// TwinCAT 3 PLC project Untitled1
// ProgramVersion: 3.1.4024.0
// libraries:
//   Tc2_MC2, * (Beckhoff Automation GmbH)
//   Tc2_Standard, * (Beckhoff Automation GmbH)
//   Tc2_System, * (Beckhoff Automation GmbH)
//   Tc2_Utilities, * (Beckhoff Automation GmbH)
//   Tc3_Module, * (Beckhoff Automation GmbH)
//   VisuDialogs, * (System)
// project tree:
//   / GlobalTextList.TcGTLO, PlcTask.TcTTO, Visualization Manager.TcVMO (not stored), VISU_TASK.TcTTO
//   POUs/ACTION/ E_ACTION_STATE.TcDUT, FB_ACTION.TcPOU, vACTION.TcVIS
//   POUs/AXES/ AXES_CYCLE.TcPOU, FB_Axis.TcPOU, GVL_AXES.TcGVL, vAXIS.TcVIS
//   POUs/EVENT_LOGGER/ E_EventType.TcDUT (not stored), FB_EventLogger.TcPOU (not stored), GVL_EVENT_LOGGER.TcGVL (not stored), ST_Event.TcDUT (not stored), UpdateEventTimestampWithSystemTime.TcPOU, UpdateTimeStamp.TcPOU, vEVENT_LOGGER.TcVIS
//   POUs/ E_STATE.TcDUT (not stored), GVL_MAIN.TcGVL, MACHINE.TcPOU, MAIN.TcPOU
//   POUs/PISTONS/ E_PISTON_STATE.TcDUT (not stored), E_PISTON_TYPE.TcDUT (not stored), FB_PISTON.TcPOU, PIST_CYCLE.TcPOU, ST_PISTON.TcDUT, vPISTONS.TcVIS, vPISTON.TcVIS (not stored)
//   POUs/STATIONS/ FB_FEEDER.TcPOU, FB_SEPARATE.TcPOU, FB_STATION.TcPOU, STATION_CYCLE.TcPOU, vFEEDER.TcVIS (not stored), vSEPARATE.TcVIS, vSTATION_CONTROLLER.TcVIS
//   VISUs/ vCOMM.TcVIS, vMACHINE.TcVIS

CONFIGURATION Untitled1
    RESOURCE PLC ON TwinCAT3
        TASK PlcTask(INTERVAL := T#10ms, PRIORITY := 20);
        TASK VISU_TASK(INTERVAL := T#200000us, PRIORITY := 30);
        PROGRAM MAIN WITH PlcTask : MAIN;
        PROGRAM VisuElems_Visu_Prg WITH VISU_TASK : VisuElems.Visu_Prg;
    END_RESOURCE
END_CONFIGURATION

// ---- POUs/ACTION/E_ACTION_STATE.TcDUT
{attribute 'qualified_only'}
{attribute 'strict'}
TYPE E_ACTION_STATE :
(
	uninit := 0,
	ready,
	done1,
	done2,
	done3,
	done4,
	done5,
	done6,
	done7,
	done8,
	done9,
	done10,
	busy,
	error
);
END_TYPE

// ---- POUs/PISTONS/ST_PISTON.TcDUT
 TYPE ST_PISTON :
STRUCT
	ePISTON_TYPE: E_PISTON_TYPE;
	nNAME: STRING;
	openTime: REAL:=5;
	closeTime: REAL:=5;
	timeoutOpen:  TIME:=T#5S;
	timeoutClose: TIME:=T#5S;
	bOPEN_BY_DEFAULT: BOOL:= FALSE;
	
	
END_STRUCT
	
END_TYPE

// ---- POUs/AXES/GVL_AXES.TcGVL
//{attribute 'qualified_only'}
VAR_GLOBAL
	
	
END_VAR

// ---- POUs/GVL_MAIN.TcGVL
//{attribute 'qualified_only'}
VAR_GLOBAL
	fbFEEDER: FB_FEEDER;
	fbSEPARATE1: FB_SEPARATE;
	fbSEPARATE2: FB_SEPARATE;
	LIFT1:FB_Axis;
	XY1:FB_Axis;
	LIFT2:FB_Axis;
	XY2:FB_Axis;
	PIST1: FB_PISTON;
	PIST2: FB_PISTON;
	PIST_FEEDER1: FB_PISTON;
	PIST_FEEDER2: FB_PISTON;
	PIST_FEEDER3: FB_PISTON;
	PIST_SEPARATE1_1: FB_PISTON;
	PIST_SEPARATE1_2: FB_PISTON;
	PIST_SEPARATE1_3: FB_PISTON;
	PIST_SEPARATE1_4: FB_PISTON;
	PIST_SEPARATE1_5: FB_PISTON;
	PIST_SEPARATE1_6: FB_PISTON;
	PIST_SEPARATE2_1: FB_PISTON;
	PIST_SEPARATE2_2: FB_PISTON;
	PIST_SEPARATE2_3: FB_PISTON;
	PIST_SEPARATE2_4: FB_PISTON;
	PIST_SEPARATE2_5: FB_PISTON;
	PIST_SEPARATE2_6: FB_PISTON;
	ACTION1:FB_ACTION;
	ACTION2:FB_ACTION;
	
	bMAIN_RESET:BOOL:=FALSE;
	iMAIN_STATE: INT:=98;
	bMAIN_PAUSE:BOOL:=FALSE;
	bMAIN_START:BOOL:=FALSE;
END_VAR

// ---- POUs/MAIN.TcPOU
PROGRAM MAIN
VAR

	
	
END_VAR



AXES_CYCLE();
PIST_CYCLE();
STATION_CYCLE();

END_PROGRAM

// ---- POUs/AXES/AXES_CYCLE.TcPOU
PROGRAM AXES_CYCLE
VAR
END_VAR

GRP1();

ACTION GRP1:
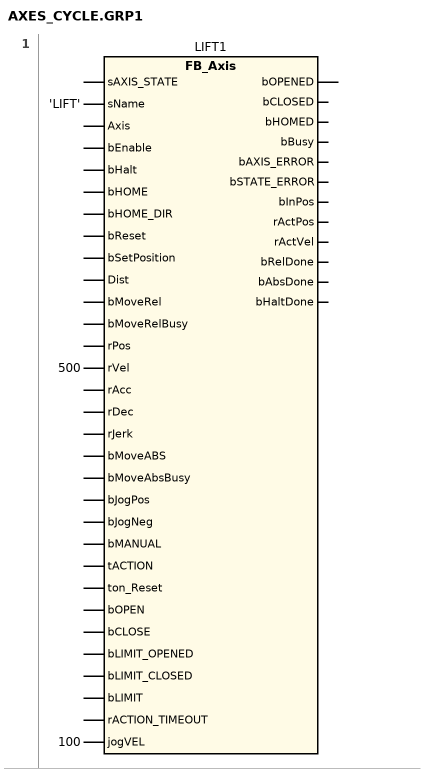
// NETWORK 1
LIFT1(sName := 'LIFT', rVel := 500, jogVEL := 100); // FB_Axis

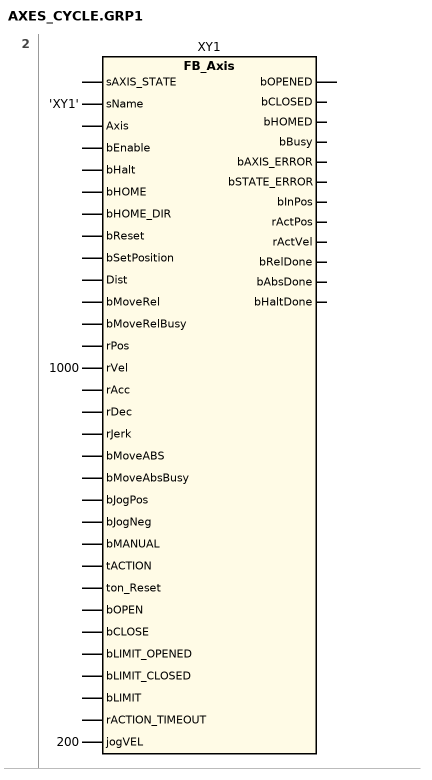
// NETWORK 2
XY1(sName := 'XY1', rVel := 1000, jogVEL := 200); // FB_Axis

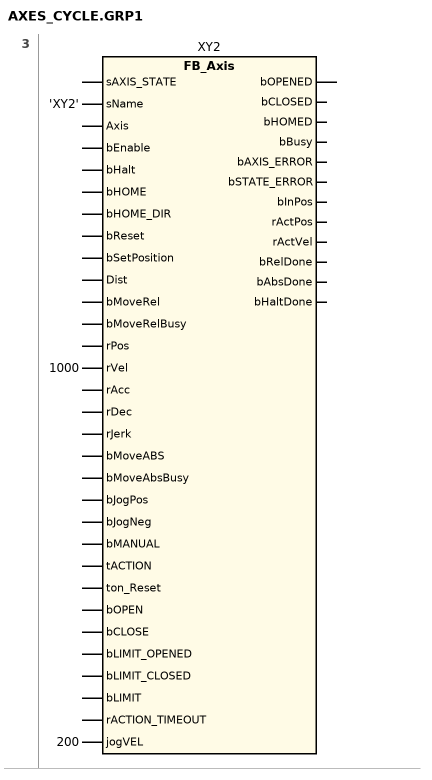
// NETWORK 3
XY2(sName := 'XY2', rVel := 1000, jogVEL := 200); // FB_Axis

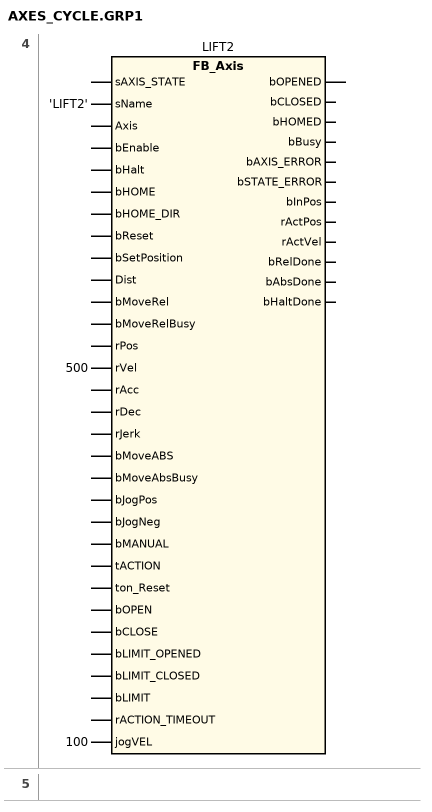
// NETWORK 4
LIFT2(sName := 'LIFT2', rVel := 500, jogVEL := 100); // FB_Axis

// NETWORK 5
END_ACTION

END_PROGRAM

// ---- POUs/AXES/FB_Axis.TcPOU
FUNCTION_BLOCK FB_Axis
VAR_INPUT
	eSTATE:E_STATE:=E_STATE.uninit;
	sAXIS_STATE:STRING:='UNINIT';
	sName:STRING;
	Axis:Axis_ref;
	bEnable:BOOL:=FALSE;
	bHalt:BOOL:=FALSE;
	bHOME:BOOL:=FALSE;
	bHOME_DIR:BOOL;
	bReset:BOOL:=FALSE;
	bSetPosition:BOOL:=FALSE;
	Dist:REAL;
	bMoveRel:BOOL:=FALSE;
	bMoveRelBusy:BOOL;
	rPos:LREAL;
	rVel:LREAL;
	rAcc:LREAL;
	rDec:LREAL;
	rJerk:LREAL;
	bMoveABS:BOOL:=FALSE;
	bMoveAbsBusy:BOOL;
	bJogPos:BOOL;
	bJogNeg:BOOL;
	bMANUAL:BOOL:=FALSE;
	tACTION:TON;
	ton_Reset: TON;
	bOPEN:BOOL;
	bCLOSE:BOOL;
	bLIMIT_OPENED:BOOL;
	bLIMIT_CLOSED:BOOL;
	bLIMIT:BOOL;
	rACTION_TIMEOUT:TIME:=T#10S;
	jogVEL: REAL;
	bSTOP:BOOL;
END_VAR

VAR_OUTPUT
	bOPENED:BOOL;
	bCLOSED:BOOL;
	bHOMED:BOOL;
	bBusy: BOOL;
	bAXIS_ERROR:BOOL;
	bSTATE_ERROR:BOOL;
	bInPos:BOOL;
	rActPos:LREAL;
	rActVel:LREAL;
	bRelDone:BOOL;
	bAbsDone:BOOL;
	bHaltDone:BOOL;
END_VAR
VAR
	bSTART_ACTION:BOOL;
	iHOME_STATE: INT:=98;
	iAXIS_STATE:INT:=98;
	tDelay: TON;
	bDelay:BOOL:=FALSE;
	MoveAbsolute: MC_MoveAbsolute;
	power: MC_Power;
	Reset: MC_Reset;
	SetPosition: MC_SetPosition;
	JOG: MC_Jog;
	RELATIVE: MC_MoveRelative;
	HALT: MC_Halt;
	HOME: MC_Home;
	bFirst_run:BOOL:=FALSE;
	bStopBusy:BOOL;
	
	
	
	
END_VAR

IF NOT bFirst_run THEN
	RESET.Execute:=TRUE;
	 bFirst_run:=TRUE;
END_IF

rActPos:=Axis.NcToPlc.ActPos;
rActVel:=Axis.NcToPlc.ActVelo;



IF RELATIVE.Busy OR JOG.Busy OR moveAbsolute.busy THEN
	bBusy:=TRUE;
END_IF
IF NOT RELATIVE.Busy AND NOT JOG.Busy AND NOT moveAbsolute.busy THEN
	bBusy:=FALSE;
END_IF

IF POWER.error OR RELATIVE.error OR MoveAbsolute.error OR JOG.error THEN
	bAXIS_ERROR:=TRUE;
END_IF
IF NOT POWER.error AND NOT RELATIVE.error AND NOT MoveAbsolute.error AND NOT JOG.error THEN
	bAXIS_ERROR:=FALSE;
END_IF

IF bRelDone OR  bAbsDone THEN
	bInPos:=TRUE;
END_IF
IF bBusy THEN
	bInPos:=FALSE;
	bRelDone:=FALSE;
	bAbsDone:=FALSE;
END_IF


CMDs();
mAXIS_STATE_MACHINE();

ACTION aAXIS_ERROR:
gEventType:= 'axis Alarm'; 
gEventSeverity:= 'Error';

gEventName:= sNAME;
IF iAXIS_STATE=1  THEN
	gEventText:='axis homing';
	gEventIdentity:=2001;
END_IF
IF iAXIS_STATE=20  THEN
	gEventText:='axis opening';
	gEventIdentity:=2002;
END_IF
IF iAXIS_STATE=40  THEN
	gEventText:='axis closing';
	gEventIdentity:=2003;
END_IF
fbEventLogger.mAdd();
END_ACTION

ACTION aHOME:
bHOME:=TRUE;
END_ACTION

METHOD clear_cmd_req : BOOL
VAR_INPUT
END_VAR

bMoveABS:= bMoveRel:= bJogPos:= bJogNeg:=FALSE;
END_METHOD

ACTION CMDs:
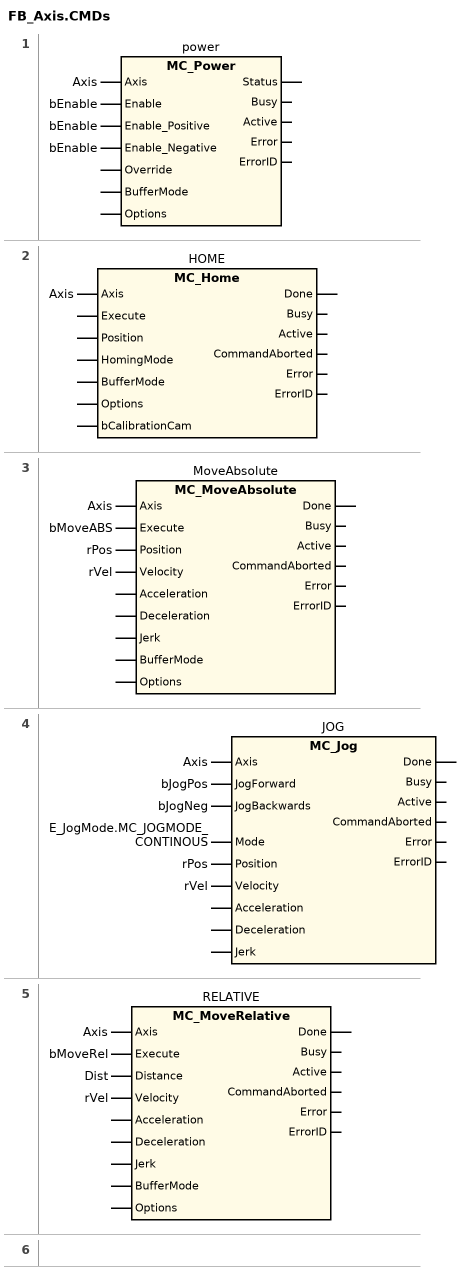
// NETWORK 1
power(Axis := Axis, Enable := bEnable, Enable_Positive := bEnable, Enable_Negative := bEnable); // MC_Power

// NETWORK 2
HOME(Axis := Axis); // MC_Home

// NETWORK 3
MoveAbsolute(Axis := Axis, Execute := bMoveABS, Position := rPos, Velocity := rVel); // MC_MoveAbsolute

// NETWORK 4
JOG(
    Axis := Axis,
    JogForward := bJogPos,
    JogBackwards := bJogNeg,
    Mode := E_JogMode.MC_JOGMODE_CONTINOUS,
    Position := rPos,
    Velocity := rVel); // MC_Jog

// NETWORK 5
RELATIVE(Axis := Axis, Execute := bMoveRel, Distance := Dist, Velocity := rVel); // MC_MoveRelative

// NETWORK 6

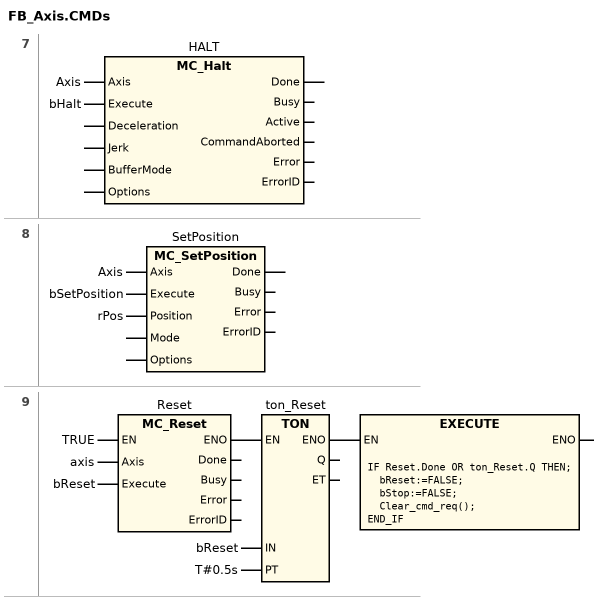
// NETWORK 7
HALT(Axis := Axis, Execute := bHalt); // MC_Halt

// NETWORK 8
SetPosition(Axis := Axis, Execute := bSetPosition, Position := rPos); // MC_SetPosition

// NETWORK 9
Reset(Axis := axis, Execute := bReset); // MC_Reset
ton_Reset(IN := bReset, PT := T#0.5s); // TON

IF Reset.Done OR ton_Reset.Q THEN;
	bReset:=FALSE;
	bStop:=FALSE;
	Clear_cmd_req();
END_IF
END_ACTION

METHOD mAXIS_STATE_MACHINE : BOOL
VAR_INPUT
	
END_VAR
tACTION(IN:= bSTART_ACTION, PT:=rACTION_TIMEOUT , Q=> , ET=> );
IF bHOME_DIR THEN
	bLIMIT:=bLIMIT_OPENED;
ELSE
	bLIMIT:=bLIMIT_CLOSED;
END_IF


CASE iAXIS_STATE OF
	1:// ============================================== HOMING
		eSTATE:=E_STATE.busy;
		bSTART_ACTION:=TRUE;
		sAXIS_STATE:='HOMING - TO SENSOR';
		bOPENED:=FALSE;bCLOSED:=FALSE;bOPEN:=FALSE;bCLOSE:=FALSE;bHOMED:=FALSE;bHOME:=FALSE;
		bENABLE:=TRUE;
		rVel:= jogVEL;
		IF bHOME_DIR THEN
			bJogPos:=TRUE;
		ELSE
			bJogNeg:=TRUE;
		END_IF
		
		IF bLIMIT THEN
			bSTART_ACTION:=FALSE;
			bJogNeg:=FALSE;
			bJogPos:=FALSE;
			iAXIS_STATE:=2;
		END_IF
		IF tACTION.Q THEN
			bSTART_ACTION:=FALSE;
			aAXIS_ERROR();
			iAXIS_STATE:=99;
			bSTATE_ERROR:=TRUE;
		END_IF
	2://FROM LIMIT
			sAXIS_STATE:= 'HOMING- FROM SENSOR';
			IF Axis.NcToPlc.ActVelo= 0 THEN
				rVel:= jogVEL/5;
				IF bHOME_DIR THEN
					bJogNeg:=TRUE;
				ELSE
					bJogPos:=TRUE;
				END_IF
				iAXIS_STATE:=3;
			END_IF	
	3:// FINISH
			IF NOT bLIMIT THEN
				bJogNeg:=FALSE;
				bJogPos:=FALSE;
				IF Axis.NcToPlc.ActVelo= 0 THEN
					bHOMED:=TRUE;
					IF bHOME_DIR THEN
						iAXIS_STATE:=100;// to ready state
						bOPENED:=TRUE;
					ELSE
						iAXIS_STATE:=100;// to ready state
						bCLOSED:=TRUE;
					END_IF
				END_IF
			END_IF
	20://=============================================== OPENING
		eSTATE:=E_STATE.busy;
		sAXIS_STATE:= 'OPENING';
		bSTART_ACTION:=TRUE;
		bOPENED:=FALSE;bCLOSED:=FALSE;bOPEN:=FALSE;bCLOSE:=FALSE;bHOMED:=FALSE;bHOME:=FALSE;
		bENABLE:=TRUE;
		rVel:= jogVEL;
		bJogPos:=TRUE;
		IF bLIMIT_OPENED THEN
			iAXIS_STATE:=21;// to deccell
			bJogPos:=FALSE;
			bSTART_ACTION:=FALSE;
		END_IF
		IF tACTION.Q THEN
			bSTART_ACTION:=FALSE;
			aAXIS_ERROR();
			iAXIS_STATE:=99;
			bSTATE_ERROR:=TRUE;
		END_IF
		
		21:
			sAXIS_STATE:= 'OPEN DECCELERATING';
			IF Axis.NcToPlc.ActVelo= 0 THEN
				iAXIS_STATE:=100;
				bOPENED:=TRUE;
			END_IF
	
	40://=============================================== CLOSING
		eSTATE:=E_STATE.busy;
		sAXIS_STATE:= 'CLOSING';
		bSTART_ACTION:=TRUE;
		bOPENED:=FALSE;bCLOSED:=FALSE;bOPEN:=FALSE;bCLOSE:=FALSE;bHOMED:=FALSE;bHOME:=FALSE;
		bENABLE:=TRUE;
		rVel:= jogVEL;
		bJogNeg:=TRUE;
		IF bLIMIT_CLOSED THEN
			iAXIS_STATE:=41;// to deccell
			bJogNeg:=FALSE;
			bSTART_ACTION:=FALSE;
		END_IF
		IF tACTION.Q THEN
			bSTART_ACTION:=FALSE;
			aAXIS_ERROR();
			iAXIS_STATE:=99;
			bSTATE_ERROR:=TRUE;
		END_IF
		
		41:
			sAXIS_STATE:= 'CLOSE DECCELERATING';
			IF Axis.NcToPlc.ActVelo= 0 THEN
				iAXIS_STATE:=100;
				bCLOSED:=TRUE;
			END_IF
	
	50:	//========================ABSOLUTE=====================
	eSTATE:=E_STATE.busy;
	sAXIS_STATE:='MOVING ABSOLUTE';
	bAbsDone:=FALSE; bOPENED:=FALSE;bCLOSED:=FALSE;bOPEN:=FALSE;bCLOSE:=FALSE;bHOMED:=FALSE;bHOME:=FALSE;
	IF moveAbsolute.Done OR HALT.Done THEN
		iAXIS_STATE:=100;
		bAbsDone:=TRUE;
		bMoveAbs:=FALSE;
	END_IF
	51://========================RELATIVE=====================
	eSTATE:=E_STATE.busy;
	sAXIS_STATE:='MOVING RELATIVE';
	bRelDone:=FALSE; bOPENED:=FALSE;bCLOSED:=FALSE;bOPEN:=FALSE;bCLOSE:=FALSE;bHOMED:=FALSE;bHOME:=FALSE;
	IF RELATIVE.Done OR HALT.Done THEN
		iAXIS_STATE:=100; 
		bRelDone:=TRUE;
		bMoveRel:=FALSE;
	END_IF
	52://======================= HALT =========================
	sAXIS_STATE:='HALTING';
	bHaltDone:=FALSE;bOPENED:=FALSE;bCLOSED:=FALSE;bOPEN:=FALSE;bCLOSE:=FALSE;bHOMED:=FALSE;bHOME:=FALSE;
	IF HALT.Done THEN
		iAXIS_STATE:=100;
		bHaltDone:=TRUE;
		bHALT:=FALSE;
	END_IF		
	98:// ============================================ UNINIT
		eSTATE:=E_STATE.uninit;
		sAXIS_STATE:='UNINIT';
		IF bHOME THEN
			iAXIS_STATE:=1;
			bSTATE_ERROR:=FALSE;
		END_IF
		
	99://======================================= ERROR 
		eSTATE:=E_STATE.error;
		sAXIS_STATE:='AXIS STATE ERROR';
		bJogNeg:=FALSE;
		bJogPos:=FALSE;
		bHOMED:=FALSE;
		IF bHOME THEN
			iAXIS_STATE:=1;
			bSTATE_ERROR:=FALSE;
		END_IF
		
	100://=============================================== READY
		eSTATE:=E_STATE.ready;
		sAXIS_STATE:='READY';
		IF bOPENED THEN
		sAXIS_STATE:= 'OPENED';
		END_IF
		IF bCLOSED THEN
		sAXIS_STATE:= 'CLOSED';
		END_IF
		IF bHOME AND NOT bHOMED THEN
			iAXIS_STATE:=1;
			bSTATE_ERROR:=FALSE;
		END_IF
		IF bCLOSE AND NOT bCLOSED THEN
			iAXIS_STATE:=40;
			bSTATE_ERROR:=FALSE;
		END_IF
		IF bOPEN AND NOT bOPENED THEN
			iAXIS_STATE:=20;
			bSTATE_ERROR:=FALSE;
		END_IF
		IF bMoveAbs THEN
			iAXIS_STATE:=50;
			bSTATE_ERROR:=FALSE;
		END_IF
		IF bMoveRel THEN
			iAXIS_STATE:=51;
			bSTATE_ERROR:=FALSE;
		END_IF
		IF bHALT THEN
			iAXIS_STATE:=52;
			bSTATE_ERROR:=FALSE;
		END_IF
	
END_CASE
END_METHOD

METHOD mMOVE_ABS : BOOL
VAR_INPUT
	movement:REAL;
END_VAR
rPOS:=movement;
bMoveAbs:=TRUE;
END_METHOD

METHOD mMOVE_REL : BOOL
VAR_INPUT
	movement:REAL;
END_VAR
Dist:=movement;
bMoveRel:=TRUE;
END_METHOD

END_FUNCTION_BLOCK

// ---- POUs/PISTONS/PIST_CYCLE.TcPOU
PROGRAM PIST_CYCLE
VAR
	bFirstRun:BOOL:=FALSE;
	counter :INT;
END_VAR


//IF NOT bFirstRun THEN
//	FOR counter:=1 TO iNUMBER_OF_PISTONS BY 1 DO
//		fbPist[counter].bInit:=1;
//	END_FOR;
//bFirstRun:=TRUE;
//END_IF
 

grp1();

ACTION grp1:
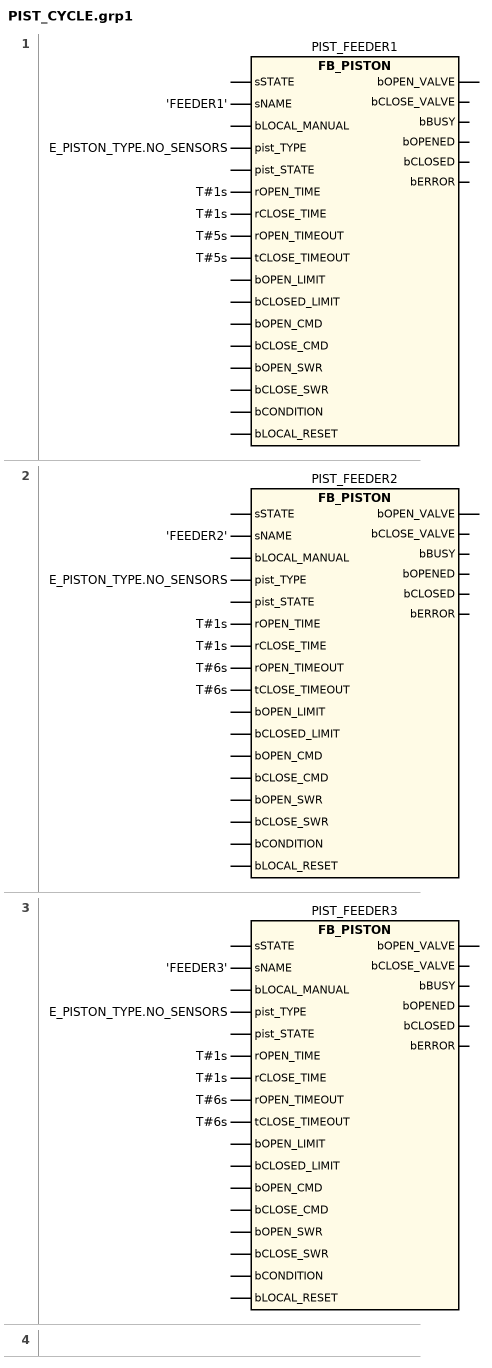
// NETWORK 1
PIST_FEEDER1(
    sNAME := 'FEEDER1',
    pist_TYPE := E_PISTON_TYPE.NO_SENSORS,
    rOPEN_TIME := T#1s,
    rCLOSE_TIME := T#1s,
    rOPEN_TIMEOUT := T#5s,
    tCLOSE_TIMEOUT := T#5s); // FB_PISTON

// NETWORK 2
PIST_FEEDER2(
    sNAME := 'FEEDER2',
    pist_TYPE := E_PISTON_TYPE.NO_SENSORS,
    rOPEN_TIME := T#1s,
    rCLOSE_TIME := T#1s,
    rOPEN_TIMEOUT := T#6s,
    tCLOSE_TIMEOUT := T#6s); // FB_PISTON

// NETWORK 3
PIST_FEEDER3(
    sNAME := 'FEEDER3',
    pist_TYPE := E_PISTON_TYPE.NO_SENSORS,
    rOPEN_TIME := T#1s,
    rCLOSE_TIME := T#1s,
    rOPEN_TIMEOUT := T#6s,
    tCLOSE_TIMEOUT := T#6s); // FB_PISTON

// NETWORK 4
END_ACTION

END_PROGRAM

// ---- POUs/PISTONS/FB_PISTON.TcPOU
FUNCTION_BLOCK FB_PISTON
VAR_INPUT
	eSTATE:E_STATE:=E_STATE.uninit;
	sSTATE:STRING:='UNINIT';
	sNAME:STRING;
	bLOCAL_MANUAL: BOOL:=FALSE;
	pist_TYPE: E_PISTON_TYPE;
	pist_STATE: E_PISTON_STATE:=E_PISTON_STATE.uninit;
	rOPEN_TIME: TIME;
	rCLOSE_TIME: TIME;
	rOPEN_TIMEOUT: TIME;
	tCLOSE_TIMEOUT: TIME;
	bOPEN_LIMIT: BOOL;
	bCLOSED_LIMIT: BOOL;
	bOPEN_CMD: BOOL;
	bCLOSE_CMD: BOOL;
	bOPEN_SWR: BOOL;
	bCLOSE_SWR: BOOL;
	bCONDITION: BOOL:=TRUE;
	bLOCAL_RESET:BOOL;
END_VAR
VAR_OUTPUT
	bOPEN_VALVE: BOOL;
	bCLOSE_VALVE: BOOL;
	bBUSY:BOOL;
	bOPENED:BOOL;
	bCLOSED:BOOL;
	bERROR:BOOL:=FALSE;
END_VAR
VAR
	T_OPEN: TON;
	T_OPEN_TIMEOUT: TON;
	T_CLOSE: TON;
	T_CLOSE_TIMEOUT: TON;
	bOPEN_DEFAULT: BOOL:=FALSE;
	bFIRST_DONE: BOOL:=FALSE;
	
END_VAR

T_OPEN(IN:= bOPEN_CMD, PT:=rOPEN_TIME , Q=> , ET=> );
T_CLOSE(IN:=  NOT bOPEN_CMD, PT:=rCLOSE_TIME , Q=> , ET=> );
T_OPEN_TIMEOUT(IN:= bOPEN_CMD , PT:= rOPEN_TIMEOUT, Q=> , ET=> );
T_CLOSE_TIMEOUT(IN:=  NOT bOPEN_CMD , PT:= tCLOSE_TIMEOUT, Q=> , ET=> );

IF bLOCAL_RESET THEN//========================== RESET================
	bLOCAL_RESET:=FALSE;
	pist_STATE:=E_PISTON_STATE.uninit;
END_IF

IF NOT bLOCAL_MANUAL THEN//====================== MANUAL ==============
	bOPEN_CMD:=bOPEN_SWR;
END_IF

IF NOT bFIRST_DONE THEN  // ============== check default mode ===============
	bFIRST_DONE:=TRUE;
	IF bOPEN_DEFAULT THEN
		bOPEN_CMD:=TRUE;
	ELSE
		bOPEN_CMD:=FALSE;
	END_IF
END_IF
//================================================== UNINIT =====================================================
CASE pist_STATE OF
	E_PISTON_STATE.uninit:
		eSTATE:=E_STATE.uninit;
		bERROR:=FALSE;
		IF bOPEN_CMD  THEN
			bOPEN_VALVE:=TRUE;
			bCLOSE_VALVE:=FALSE;
			pist_STATE:=E_PISTON_STATE.opening;
		ELSE
			bOPEN_VALVE:=FALSE;
			bCLOSE_VALVE:=TRUE;
			pist_STATE:=E_PISTON_STATE.closing;
		END_IF
//================================================== OPENING =====================================================
	E_PISTON_STATE.opening:
	eSTATE:=E_STATE.busy;
	sSTATE:='OPENING';
	bBUSY:=TRUE; bOPENED:=FALSE; bCLOSED:=FALSE;
	CASE pist_TYPE OF//------------------------------no sensors
		E_PISTON_TYPE.NO_SENSORS:
		IF T_OPEN.Q THEN
			pist_STATE:=E_PISTON_STATE.opened;
		END_IF
		//----------------------------- both sensors
		E_PISTON_TYPE.BOTH:
		IF bOPEN_LIMIT THEN
			pist_STATE:=E_PISTON_STATE.opened;
		END_IF
		IF T_OPEN_TIMEOUT.Q THEN
			bOPEN_CMD:=FALSE;
			aPISTON_ERROR();
			pist_STATE:=E_PISTON_STATE.error;
		END_IF
		//----------------------------- only open sensor
		E_PISTON_TYPE.ONLY_OPEN:
		IF bOPEN_LIMIT THEN
			pist_STATE:=E_PISTON_STATE.opened;
		END_IF
		IF T_OPEN_TIMEOUT.Q THEN
			bOPEN_CMD:=FALSE;
			aPISTON_ERROR();
			pist_STATE:=E_PISTON_STATE.error;
		END_IF
		//----------------------------- only close sensor
		E_PISTON_TYPE.ONLY_CLOSE:
		IF T_OPEN.Q THEN
			pist_STATE:=E_PISTON_STATE.opened;
		END_IF
	END_CASE
//================================================== CLOSING =====================================================	
	E_PISTON_STATE.closing:
	eSTATE:=E_STATE.busy;
	sSTATE:='CLOSING'; bOPENED:=FALSE; bCLOSED:=FALSE;
	bBUSY:=TRUE;
	CASE pist_TYPE OF//--------------------------------------- no sensors
		E_PISTON_TYPE.NO_SENSORS:
		IF T_CLOSE.Q THEN
			pist_STATE:=E_PISTON_STATE.closed;
		END_IF
		//-------------------------------------- both sensors
		E_PISTON_TYPE.BOTH:
		IF bCLOSED_LIMIT THEN
			pist_STATE:=E_PISTON_STATE.closed;
		END_IF
		IF T_CLOSE_TIMEOUT.Q THEN
			bOPEN_CMD:=TRUE;
			pist_STATE:=E_PISTON_STATE.error;
		END_IF
		//-------------------------------------- only close sensor
		E_PISTON_TYPE.ONLY_CLOSE:
		IF bCLOSED_LIMIT THEN
			pist_STATE:=E_PISTON_STATE.closed;
		END_IF
		IF T_CLOSE_TIMEOUT.Q THEN
			bOPEN_CMD:=TRUE;
			aPISTON_ERROR();
			pist_STATE:=E_PISTON_STATE.error;
		END_IF
		//----------------------------- only close sensor
		E_PISTON_TYPE.ONLY_OPEN:
		IF T_CLOSE.Q THEN
			pist_STATE:=E_PISTON_STATE.closed;
		END_IF
	END_CASE
//================================================== OPENED =====================================================	
	E_PISTON_STATE.opened:
	eSTATE:=E_STATE.ready;
	sSTATE:='OPENED';
	bBUSY:=FALSE; bOPENED:=TRUE; bCLOSED:=FALSE;
	IF NOT bOPEN_CMD  THEN
		pist_STATE:=E_PISTON_STATE.closing;
		bOPEN_VALVE:=FALSE;
		bCLOSE_VALVE:=TRUE;
	END_IF
	CASE pist_TYPE OF
		//-------------------------------------- both sensors
		E_PISTON_TYPE.BOTH:
		IF NOT bOPEN_LIMIT THEN
			bOPEN_CMD:=FALSE;
			aPISTON_ERROR();
			pist_STATE:=E_PISTON_STATE.error;
		END_IF
		//-------------------------------------- only open sensor
		E_PISTON_TYPE.ONLY_OPEN:
		IF NOT bOPEN_LIMIT THEN
			bOPEN_CMD:=FALSE;
			aPISTON_ERROR();
			pist_STATE:=E_PISTON_STATE.error;
		END_IF
	END_CASE
//================================================== CLOSED =====================================================	
	E_PISTON_STATE.closed:
	eSTATE:=E_STATE.ready;
	sSTATE:='CLOSED';
	bBUSY:=FALSE; bOPENED:=FALSE; bCLOSED:=TRUE;
	IF bOPEN_CMD  THEN
		pist_STATE:=E_PISTON_STATE.opening;
		bOPEN_VALVE:=TRUE;
		bCLOSE_VALVE:=FALSE;
	END_IF
	CASE pist_TYPE OF
		//-------------------------------------- both sensors
		E_PISTON_TYPE.BOTH:
		IF NOT bCLOSED_LIMIT THEN
			bOPEN_CMD:=TRUE;
			aPISTON_ERROR();
			pist_STATE:=E_PISTON_STATE.error;
		END_IF
		//-------------------------------------- only close sensor
		E_PISTON_TYPE.ONLY_CLOSE:
		IF NOT bCLOSED_LIMIT THEN
			bOPEN_CMD:=TRUE;
			aPISTON_ERROR();
			pist_STATE:=E_PISTON_STATE.error;
		END_IF
	END_CASE
//================================================== ERROR =====================================================	
	E_PISTON_STATE.error:
	eSTATE:=E_STATE.error;
	sSTATE:='ERROR';
	bERROR:=TRUE;
	//
END_CASE

ACTION aCLOSE:
bOPEN_SWR:=FALSE;
END_ACTION

ACTION aHOME:
IF bOPEN_DEFAULT THEN
	bOPEN_SWR:=TRUE;
ELSE
	bOPEN_SWR:=FALSE;
END_IF
END_ACTION

ACTION aOPEN:
bOPEN_SWR:=TRUE;
END_ACTION

ACTION aPISTON_ERROR:
gEventType:= 'piston Alarm'; 
gEventSeverity:= 'Error';

gEventName:= sNAME;
IF pist_STATE=E_PISTON_STATE.opening  THEN
	gEventText:='piston opening';
	gEventIdentity:=1001;
END_IF
IF pist_STATE=E_PISTON_STATE.closing THEN
	gEventText:='piston closing';
	gEventIdentity:=1002;
END_IF
IF pist_STATE=E_PISTON_STATE.closed THEN
	gEventText:='piston closed';
	gEventIdentity:=1003;
END_IF
IF pist_STATE=E_PISTON_STATE.opened THEN
	gEventText:='piston opened';
	gEventIdentity:=1004;
END_IF
fbEventLogger.mAdd();
END_ACTION

ACTION aRESET:
bLOCAL_RESET:=TRUE;
END_ACTION

END_FUNCTION_BLOCK

// ---- POUs/STATIONS/STATION_CYCLE.TcPOU
PROGRAM STATION_CYCLE
VAR
END_VAR

grp_feeder();
grp_separate();

ACTION grp_feeder:
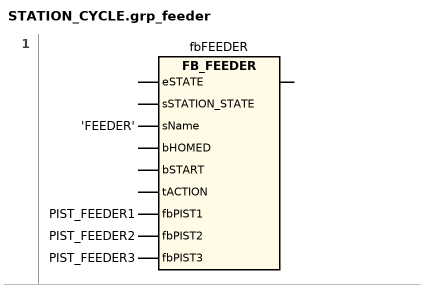
// NETWORK 1
fbFEEDER(sName := 'FEEDER', fbPIST1 := PIST_FEEDER1, fbPIST2 := PIST_FEEDER2, fbPIST3 := PIST_FEEDER3); // FB_FEEDER
END_ACTION

ACTION grp_separate:
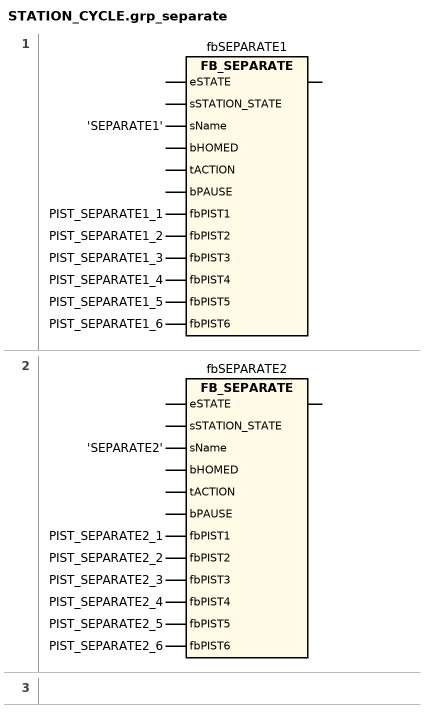
// NETWORK 1
fbSEPARATE1(
    sName := 'SEPARATE1',
    fbPIST1 := PIST_SEPARATE1_1,
    fbPIST2 := PIST_SEPARATE1_2,
    fbPIST3 := PIST_SEPARATE1_3,
    fbPIST4 := PIST_SEPARATE1_4,
    fbPIST5 := PIST_SEPARATE1_5,
    fbPIST6 := PIST_SEPARATE1_6); // FB_SEPARATE

// NETWORK 2
fbSEPARATE2(
    sName := 'SEPARATE2',
    fbPIST1 := PIST_SEPARATE2_1,
    fbPIST2 := PIST_SEPARATE2_2,
    fbPIST3 := PIST_SEPARATE2_3,
    fbPIST4 := PIST_SEPARATE2_4,
    fbPIST5 := PIST_SEPARATE2_5,
    fbPIST6 := PIST_SEPARATE2_6); // FB_SEPARATE

// NETWORK 3
END_ACTION

END_PROGRAM

// ---- POUs/STATIONS/FB_FEEDER.TcPOU
FUNCTION_BLOCK FB_FEEDER EXTENDS FB_STATION
VAR_INPUT
	fbPIST1: REFERENCE TO FB_PISTON;
	fbPIST2: REFERENCE TO FB_PISTON;
	fbPIST3: REFERENCE TO FB_PISTON;
	rACTION_TIME: TIME;
	bTEST:BOOL;
END_VAR
VAR_OUTPUT
END_VAR
VAR
	bSTART_ACTION:BOOL;
	
END_VAR

tACTION(IN:= bSTART_ACTION, PT:=rACTION_TIME , Q=> , ET=> );
IF bRESET THEN
	iSTATION_STATE:=98 ;
	bPAUSE:=FALSE;
END_IF

CASE iSTATION_STATE OF 
	1: //open pist 1
		eSTATE:=E_STATE.busy;
		sSTATION_STATE:=' PIST1 OPENING';
		fbPIST1.aOPEN();
		IF fbPIST1.eSTATE= E_STATE.busy THEN
			iSTATION_STATE:=2;
		END_IF
	2://wait for pist1 ready
		IF fbPIST1.eSTATE= E_STATE.ready THEN
			IF NOT bPAUSE THEN
				iSTATION_STATE:=3;
			END_IF
		END_IF
		IF PIST1.eSTATE= E_STATE.error THEN
			iSTATION_STATE:=99;
		END_IF
	3:	//open pist 2
		sSTATION_STATE:=' PIST2 OPENING';
		fbPIST2.aOPEN();
		IF fbPIST2.eSTATE= E_STATE.busy THEN
			iSTATION_STATE:=4;
		END_IF
	4:
		IF fbPIST2.eSTATE= E_STATE.ready THEN
			IF NOT bPAUSE THEN
				iSTATION_STATE:=5;
			END_IF
		END_IF
		IF fbPIST2.eSTATE= E_STATE.error THEN
			iSTATION_STATE:=99;
		END_IF
	5:	//open pist 3
		sSTATION_STATE:=' PIST3 OPENING';
		fbPIST3.aOPEN();
		IF fbPIST3.eSTATE= E_STATE.busy THEN
			iSTATION_STATE:=6;
		END_IF
	6:
		IF fbPIST3.eSTATE= E_STATE.ready THEN
			IF NOT bPAUSE THEN
				iSTATION_STATE:=100;
			END_IF
		END_IF
		IF fbPIST3.eSTATE= E_STATE.error THEN
			iSTATION_STATE:=99;
		END_IF

	98:
		eSTATE:=E_STATE.uninit;
		sSTATION_STATE:='UNINIT';
		bRESET:=FALSE;
		fbPIST1.aRESET();
		fbPIST2.aRESET();
		fbPIST3.aRESET();
		IF fbPIST1.eSTATE = E_STATE.uninit AND fbPIST1.eSTATE = E_STATE.uninit AND fbPIST1.eSTATE = E_STATE.uninit THEN
			iSTATION_STATE:=980;
		END_IF
	980: 
		IF fbPIST1.eSTATE= E_STATE.ready AND fbPIST2.eSTATE= E_STATE.ready AND fbPIST3.eSTATE= E_STATE.ready THEN
			iSTATION_STATE:=100;
		END_IF
		
		IF fbPIST1.bERROR OR fbPIST2.bERROR OR fbPIST3.bERROR THEN
			iSTATION_STATE:=99;
		END_IF
	
	99:
		eSTATE:=E_STATE.error;
		sSTATION_STATE:='PISTON ERROR';
		
	100:
		eSTATE:=E_STATE.ready;
		sSTATION_STATE:='READY';
		IF bSTART THEN
			bSTART:=FALSE;
			iSTATION_STATE:=1;
		END_IF
		
END_CASE

END_FUNCTION_BLOCK

// ---- POUs/STATIONS/FB_STATION.TcPOU
FUNCTION_BLOCK FB_STATION
VAR_INPUT
	eSTATE:E_STATE:=E_STATE.uninit;
	sSTATION_STATE:STRING:='UNINIT';
	sName:STRING;
	bHOMED : BOOL:=FALSE;
	tACTION:TON;
	bPAUSE:BOOL:=FALSE;
	
END_VAR
VAR_OUTPUT
END_VAR
VAR
	
	bRESET:BOOL;
	bSTART:BOOL:=FALSE;
	iSTATION_STATE:INT:=98;;
	bFIRST_RUB:BOOL:=FALSE;
END_VAR

ACTION aSTART:
bSTART:=TRUE;
END_ACTION

END_FUNCTION_BLOCK

// ---- POUs/STATIONS/FB_SEPARATE.TcPOU
FUNCTION_BLOCK FB_SEPARATE  EXTENDS FB_STATION
VAR_INPUT
	fbPIST1: REFERENCE TO FB_PISTON;
	fbPIST2: REFERENCE TO FB_PISTON;
	fbPIST3: REFERENCE TO FB_PISTON;
	fbPIST4: REFERENCE TO FB_PISTON;
	fbPIST5: REFERENCE TO FB_PISTON;
	fbPIST6: REFERENCE TO FB_PISTON;
	
END_VAR
VAR_OUTPUT
END_VAR
VAR
END_VAR

IF bRESET THEN
	iSTATION_STATE:=98 ;
	bPAUSE:=FALSE;
END_IF

CASE iSTATION_STATE OF 
	1: //open pist 1
		eSTATE:=E_STATE.busy;
		sSTATION_STATE:=' PIST1 OPENING';
		fbPIST1.aOPEN();
		IF fbPIST1.eSTATE= E_STATE.busy THEN
			iSTATION_STATE:=2;
		END_IF
	2://wait for pist1 ready
		IF fbPIST1.eSTATE= E_STATE.ready THEN
			IF NOT bPAUSE THEN
				iSTATION_STATE:=3;
			END_IF
		END_IF
		IF PIST1.eSTATE= E_STATE.error THEN
			iSTATION_STATE:=99;
		END_IF
	3:	//open pist 2
		sSTATION_STATE:=' PIST2 OPENING';
		fbPIST2.aOPEN();
		IF fbPIST2.eSTATE= E_STATE.busy THEN
			iSTATION_STATE:=4;
		END_IF
	4:
		IF fbPIST2.eSTATE= E_STATE.ready THEN
			IF NOT bPAUSE THEN
				iSTATION_STATE:=5;
			END_IF
		END_IF
		IF fbPIST2.eSTATE= E_STATE.error THEN
			iSTATION_STATE:=99;
		END_IF
	5:	//open pist 3
		sSTATION_STATE:=' PIST3 OPENING';
		fbPIST3.aOPEN();
		IF fbPIST3.eSTATE= E_STATE.busy THEN
			iSTATION_STATE:=6;
		END_IF
	6:
		IF fbPIST3.eSTATE= E_STATE.ready THEN
			IF NOT bPAUSE THEN
				iSTATION_STATE:=100;
			END_IF
		END_IF
		IF fbPIST3.eSTATE= E_STATE.error THEN
			iSTATION_STATE:=99;
		END_IF

	98:
		eSTATE:=E_STATE.uninit;
		sSTATION_STATE:='UNINIT';
		bRESET:=FALSE;
		fbPIST1.aRESET();
		fbPIST2.aRESET();
		fbPIST3.aRESET();
		IF fbPIST1.eSTATE = E_STATE.uninit AND fbPIST1.eSTATE = E_STATE.uninit AND fbPIST1.eSTATE = E_STATE.uninit THEN
			iSTATION_STATE:=980;
		END_IF
	980: 
		IF fbPIST1.eSTATE= E_STATE.ready AND fbPIST2.eSTATE= E_STATE.ready AND fbPIST3.eSTATE= E_STATE.ready THEN
			iSTATION_STATE:=100;
		END_IF
		
		IF fbPIST1.bERROR OR fbPIST2.bERROR OR fbPIST3.bERROR THEN
			iSTATION_STATE:=99;
		END_IF
	
	99:
		eSTATE:=E_STATE.error;
		sSTATION_STATE:='PISTON ERROR';
		
	100:
		eSTATE:=E_STATE.ready;
		sSTATION_STATE:='READY';
		IF bSTART THEN
			bSTART:=FALSE;
			iSTATION_STATE:=1;
		END_IF
		
END_CASE

END_FUNCTION_BLOCK

// ---- POUs/ACTION/FB_ACTION.TcPOU
FUNCTION_BLOCK FB_ACTION
VAR_INPUT
	sNAME: STRING;
	PIST: REFERENCE TO FB_PISTON;
	aLIFT:REFERENCE TO FB_Axis;
	aXY:REFERENCE TO FB_Axis;
	bSTART_OPEN:BOOL;
	bSTART_CLOSE:BOOL;
	bSTART_HOMING:BOOL;
	iHOME_STATE:INT:=98;
	iOPEN_STATE:INT:=98;
	iCLOSE_STATE:INT:=98;
	bHOME_ALL:BOOL;
	bOPEN_ALL:BOOL;
	bCLOSE_ALL:BOOL;
	tACTION:TON;
	rACTION_TIMEOUT:TIME:=T#20S;
	tHOMING:TON;
	rHOMING_TIMEOUT: TIME:=T#20S;
	tOPEN:TON;
	rOPEN_TIMEOUT: TIME:=T#20S;
	tCLOSE:TON;
	rCLOSE_TIMEOUT: TIME:=T#20S;
END_VAR
VAR_OUTPUT
	sACTION_STATE:STRING:='UNINIT';
	bSTART_ACTION:BOOL;
	iACTION_STATE:INT:=98;
	bACTION_ERROR:BOOL;
	bALL_HOMED:BOOL;
	bALL_OPENED:BOOL;
	bALL_CLOSED:BOOL;
END_VAR
VAR
END_VAR

mACTION_STATE_MACHINE();
IF bALL_HOMED THEN
	IF NOT aLIFT.bHOMED OR NOT aXY.bHOMED THEN
		bALL_HOMED:=FALSE;
		iACTION_STATE:=98;
	END_IF
END_IF

ACTION aACTION_ERROR:
gEventType:= 'action Alarm'; 
gEventSeverity:= 'Error';

gEventName:= sNAME;
IF iACTION_STATE=2  THEN
	gEventText:='action XY homing';
	gEventIdentity:=5001;
END_IF
IF iACTION_STATE=2  THEN
	gEventText:='action LIFT homing';
	gEventIdentity:=5002;
END_IF
IF iACTION_STATE=5  THEN
	gEventText:='action PISTON homing';
	gEventIdentity:=5003;
END_IF
//---------------------------------------------------
IF iACTION_STATE=14  THEN
	gEventText:='action XY opening';
	gEventIdentity:=5011;
END_IF
IF iACTION_STATE=12  THEN
	gEventText:='action LIFT opening';
	gEventIdentity:=5012;
END_IF
IF iACTION_STATE=10  THEN
	gEventText:='action PISTON opening';
	gEventIdentity:=5013;
END_IF
//---------------------------------------------------
IF iACTION_STATE=32  THEN
	gEventText:='action XY closing';
	gEventIdentity:=5021;
END_IF
IF iACTION_STATE=34  THEN
	gEventText:='action LIFT closing';
	gEventIdentity:=5022;
END_IF
IF iACTION_STATE=35  THEN
	gEventText:='action PISTON closing';
	gEventIdentity:=5023;
END_IF
fbEventLogger.mAdd();
END_ACTION

METHOD mACTION_STATE_MACHINE : BOOL
VAR_INPUT
END_VAR
tACTION(IN:= bSTART_ACTION, PT:=rACTION_TIMEOUT , Q=> , ET=> );

CASE iACTION_STATE OF
	
	1://======================================  HOME ALL	
		//HOME XY
		sACTION_STATE:='HOMING ALL XY';
		bHOME_ALL:=FALSE; bALL_HOMED:=FALSE;bALL_OPENED:=FALSE;bOPEN_ALL:=FALSE;bALL_CLOSED:=FALSE;bCLOSE_ALL:=FALSE;
		aXY.bHome:=TRUE;
		bSTART_ACTION:=TRUE;
		iACTION_STATE:=2; 
	2:
		aXY.bHome:=FALSE;
		IF aXY.bHOMED THEN
			bSTART_ACTION:=FALSE;
			iACTION_STATE:=3;
		END_IF
		IF aXY.bSTATE_ERROR THEN
			iACTION_STATE:=99;
			aACTION_ERROR();
			bSTART_ACTION:=FALSE;
			bACTION_ERROR:=TRUE;
		END_IF
			
	3://HOME LIFT
		sACTION_STATE:='HOMING ALL LIFT';
		aLIFT.bHome:=TRUE;
		bSTART_ACTION:=TRUE;
		iACTION_STATE:=4;
	4:
		aLIFT.bHome:=FALSE;
		IF aLIFT.bHOMED THEN
			bSTART_ACTION:=FALSE;
			iACTION_STATE:=5;
		END_IF
		IF aLIFT.bSTATE_ERROR THEN
			aACTION_ERROR();
			iACTION_STATE:=99;
			bSTART_ACTION:=FALSE;
			bACTION_ERROR:=TRUE;
		END_IF
	5://HOME PISTON
		sACTION_STATE:='HOMING ALL PISTON';
		bSTART_ACTION:=TRUE;
		PIST.bOPEN_SWR:=FALSE;
		IF PIST.bCLOSED THEN
			bSTART_ACTION:=FALSE;
			iACTION_STATE:=100;
			bALL_HOMED:=TRUE;
		END_IF
		IF PIST.bERROR THEN
			aACTION_ERROR();
			iACTION_STATE:=99;
			bSTART_ACTION:=FALSE;
			bACTION_ERROR:=TRUE;
		END_IF
	10://===================================== OPENING ALL
		//OPEN PISTON
		bHOME_ALL:=FALSE; bALL_HOMED:=FALSE;bALL_OPENED:=FALSE;bOPEN_ALL:=FALSE;bALL_CLOSED:=FALSE;bCLOSE_ALL:=FALSE;
		sACTION_STATE:='OPENING ALL PISTON';
		bSTART_ACTION:=TRUE;
		PIST.bOPEN_SWR:=TRUE;
		IF PIST.bOPENED THEN
			bSTART_ACTION:=FALSE;
			iACTION_STATE:=11;
		END_IF
		IF PIST.bERROR THEN
			aACTION_ERROR();
			iACTION_STATE:=99;
			bSTART_ACTION:=FALSE;
			bACTION_ERROR:=TRUE;
		END_IF
	11://OPEN LIFT
		sACTION_STATE:='OPENING ALL LIFT';
		aLIFT.bOPEN:=TRUE;
		bSTART_ACTION:=TRUE;
		iACTION_STATE:=12;
	12:
		aLIFT.bOPEN:=FALSE;
		IF aLIFT.bOPENED THEN
			bSTART_ACTION:=FALSE;
			iACTION_STATE:=13;
		END_IF
		IF aLIFT.bSTATE_ERROR THEN
			aACTION_ERROR();
			iACTION_STATE:=99;
			bSTART_ACTION:=FALSE;
			bACTION_ERROR:=TRUE;
		END_IF
	13://OPEN ALL XY
		sACTION_STATE:='OPENING ALL XY';
		aXY.bOPEN:=TRUE;
		bSTART_ACTION:=TRUE;
		iACTION_STATE:=14; 
	14:
		aXY.bOPEN:=FALSE;
		IF aXY.bOPENED THEN
			bSTART_ACTION:=FALSE;
			bALL_OPENED:=TRUE;
			iACTION_STATE:=20;
		END_IF
		IF aXY.bSTATE_ERROR THEN
			aACTION_ERROR();
			iACTION_STATE:=99;
			bSTART_ACTION:=FALSE;
			bACTION_ERROR:=TRUE;
		END_IF	

	20:// ==================================== OPENED
		sACTION_STATE:='OPENED';
		IF bCLOSE_ALL THEN
			iACTION_STATE:=30;
			bACTION_ERROR:=FALSE;
		END_IF
		IF bHOME_ALL THEN
			iACTION_STATE:=1;
			bACTION_ERROR:=FALSE;
		END_IF
		
	30://===================================== CLOSING ALL XY
		sACTION_STATE:='CLOSING ALL XY';
		bHOME_ALL:=FALSE; bALL_HOMED:=FALSE;bALL_OPENED:=FALSE;bOPEN_ALL:=FALSE;bALL_CLOSED:=FALSE;bCLOSE_ALL:=FALSE;
		aXY.bCLOSE:=TRUE;
		bSTART_ACTION:=TRUE;
		iACTION_STATE:=32; 
	32:
		aXY.bCLOSE:=FALSE;
		IF aXY.bCLOSED THEN
			bSTART_ACTION:=FALSE;
			iACTION_STATE:=33;
		END_IF
		IF aXY.bSTATE_ERROR THEN
			aACTION_ERROR();
			iACTION_STATE:=99;
			bSTART_ACTION:=FALSE;
			bACTION_ERROR:=TRUE;
		END_IF	
	33://HOME LIFT
		sACTION_STATE:='CLOSING ALL LIFT';
		aLIFT.bCLOSE:=TRUE;
		bSTART_ACTION:=TRUE;
		iACTION_STATE:=34;
	34:
		aLIFT.bCLOSE:=FALSE;
		IF aLIFT.bCLOSED THEN
			bSTART_ACTION:=FALSE;
			iACTION_STATE:=35;
		END_IF
		IF aLIFT.bSTATE_ERROR THEN
			aACTION_ERROR();
			iACTION_STATE:=99;
			bSTART_ACTION:=FALSE;
			bACTION_ERROR:=TRUE;
		END_IF
	35://CLOSE ALL PISTON
		sACTION_STATE:='CLOSING ALL PISTON';
		bSTART_ACTION:=TRUE;
		PIST.bOPEN_SWR:=FALSE;
		IF PIST.bCLOSED THEN
			bSTART_ACTION:=FALSE;
			iACTION_STATE:=40;
			bALL_CLOSED:=TRUE;
		END_IF
		IF PIST.bERROR THEN
			aACTION_ERROR();
			iACTION_STATE:=99;
			bSTART_ACTION:=FALSE;
			bACTION_ERROR:=TRUE;
		END_IF 
	40:// ==================================== CLOSED
		sACTION_STATE:='CLOSED';
		IF bOPEN_ALL THEN
			iACTION_STATE:=10;
			bACTION_ERROR:=FALSE;
		END_IF		
		IF bHOME_ALL THEN
			iACTION_STATE:=1;
			bACTION_ERROR:=FALSE;
		END_IF
		
	98://===================================== UNINIT
		sACTION_STATE:='UNINIT';
		IF bHOME_ALL THEN
			iACTION_STATE:=1;
			bACTION_ERROR:=FALSE;
		END_IF
		
	99://===================================== ERROR
		sACTION_STATE:='ERROR';
		IF bHOME_ALL THEN
			iACTION_STATE:=1;
			bACTION_ERROR:=FALSE;
		END_IF
	
	100://===================================== HOMED
		sACTION_STATE:='HOMED';
		IF bHOME_ALL THEN
			iACTION_STATE:=1;
			bACTION_ERROR:=FALSE;
		END_IF	
		IF bOPEN_ALL THEN
			iACTION_STATE:=10;
			bACTION_ERROR:=FALSE;
		END_IF
	
	
END_CASE
END_METHOD

END_FUNCTION_BLOCK

// ---- POUs/EVENT_LOGGER/UpdateEventTimestampWithSystemTime.TcPOU
FUNCTION UpdateEventTimestampWithSystemTime 
VAR_INPUT
	stEvent: REFERENCE TO ST_Event;  
	
END_VAR
VAR
	fbGETSYSTEMTIME : GETSYSTEMTIME;
	stFileTime : T_FILETIME;
END_VAR

fbGETSYSTEMTIME(timeLoDW =>stFileTime.dwLowDateTime ,
				timeHiDW =>stFileTime.dwHighDateTime );
				
stEvent.dtTimestamp:= FILETIME_TO_DT(fileTime := stFileTime);

END_FUNCTION

// ---- POUs/EVENT_LOGGER/UpdateTimeStamp.TcPOU
FUNCTION UpdateTimeStamp 
VAR_INPUT
	stUser : REFERENCE TO ST_USER;
END_VAR
VAR
	fbGETSYSTEMTIME : GETSYSTEMTIME;
	
	stFileTime : T_FILETIME;
END_VAR


fbGETSYSTEMTIME(timeLoDW =>stFileTime.dwLowDateTime ,
				timeHiDW =>stFileTime.dwHighDateTime );
				
stUser.dtTIME_STAMP:= FILETIME_TO_DT(fileTime := stFileTime);

END_FUNCTION

// ---- POUs/MACHINE.TcPOU
PROGRAM MACHINE
VAR
END_VAR



IF bMAIN_RESET THEN
	iMAIN_STATE:=98 ;
	bMAIN_PAUSE:=FALSE;
END_IF

END_PROGRAM

// ---- GlobalTextList.TcGTLO
TEXTLIST GlobalTextList
  450 = '%.2f'
  859 = '%d'
  952 = '%s'
  396 = 'ACC'
  188 = 'BUSY'
  997 = 'CLOSE'
  513 = 'CLOSE ALL'
  293 = 'CLOSED LIMIT'
  446 = 'DIST'
  904 = 'ENABLE'
  50 = 'ERROR'
  182 = 'ESTOP'
  810 = 'FEEDER'
  288 = 'GO ABS'
  776 = 'GO REL'
  373 = 'HALT'
  598 = 'HOME'
  825 = 'HOME_ALL'
  512 = 'INPOS'
  837 = 'JERK'
  268 = 'JOG +'
  202 = 'JOG -'
  309 = 'MACHINE'
  412 = 'MANUAL'
  189 = 'OPEN'
  149 = 'OPEN ALL'
  299 = 'OPENED LIMIT'
  569 = 'PAUSE'
  282 = 'PAUSED:'
  425 = 'POS'
  390 = 'Pos: %.2f'
  563 = 'POWER'
  793 = 'POWER BY STRIX'
  507 = 'R'
  779 = 'RESET'
  830 = 'SET'
  487 = 'START'
  506 = 'STRIX1200'
  245 = 'TAMAR 20MM'
  964 = 'VEL'
  60 = 'Vel: %.2f'
END_TEXTLIST

// ---- POUs/ACTION/vACTION.TcVIS
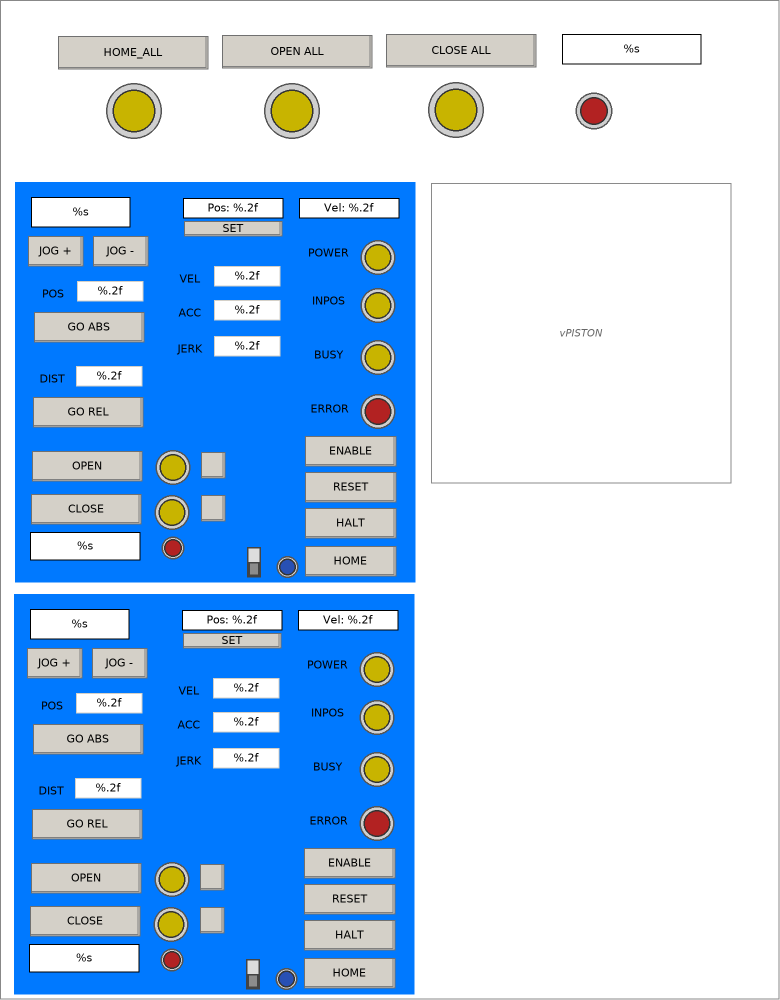
VISUALIZATION vACTION  // 780x1000
VAR_IN_OUT
	vACTION:FB_ACTION;
END_VAR
    Frame (15,182 400x400)
        shows vAXIS(vAxis := vACTION.aLIFT)
    Frame (431,183 300x300)
        shows vPISTON(PIST1 := vACTION.PIST)
    Frame (14,594 400x400)
        shows vAXIS(vAxis := vACTION.aXY)
    Button (58,36 150x33), "HOME_ALL"
        OnMouseDown: execute { vACTION.bHOME_ALL:=TRUE; }
    Lamp1 (102,79 64x64), variable: vACTION.bALL_HOMED, style: Lamp-Lamp1-Yellow
    Button (222,35 150x33), "OPEN ALL"
        OnMouseDown: execute { vACTION.bOPEN_ALL:=TRUE; }
    Lamp1 (260,79 64x64), variable: vACTION.bALL_OPENED, style: Lamp-Lamp1-Yellow
    Button (386,34 150x33), "CLOSE ALL"
        OnMouseDown: execute { vACTION.bCLOSE_ALL:=TRUE; }
    Lamp1 (424,78 64x64), variable: vACTION.bALL_CLOSED, style: Lamp-Lamp1-Yellow
    Lamp1 (573,88 42x46), variable: vACTION.bACTION_ERROR, style: Lamp-Lamp1-Red
    Rectangle (562,34 139x30), "%s", text variable: vACTION.sACTION_STATE
END_VISUALIZATION

// ---- POUs/AXES/vAXIS.TcVIS
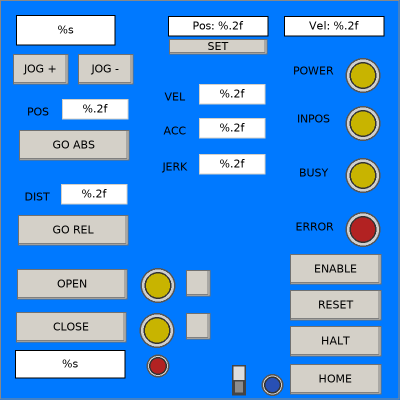
VISUALIZATION vAXIS  // 400x400
VAR_IN_OUT
	vAxis:FB_Axis;
END_VAR
    Rectangle (168,16 100x20), "Pos: %.2f", text variable: vAxis.rActPos
    Rectangle (284,16 100x20), "Vel: %.2f", text variable: vAxis.rActVel
    Lamp1 (343,53 40x45), variable: vAxis.power.Enable, style: Lamp-Lamp1-Yellow
    Label (286,60 55x22), "POWER"
    Lamp1 (343,101 40x45), variable: vAxis.bInPos, style: Lamp-Lamp1-Yellow
    Lamp1 (343,207 40x45), variable: vAxis.bAXIS_ERROR, style: Lamp-Lamp1-Red
    Lamp1 (343,153 40x45), variable: vAxis.bBusy, style: Lamp-Lamp1-Yellow
    Label (286,108 55x22), "INPOS"
    Label (287,216 55x22), "ERROR"
    Label (286,162 55x22), "BUSY"
    Button (290,254 91x30), "ENABLE"
        toggle vAxis.bEnable
    Button (290,290 91x30), "RESET"
        toggle vAxis.bReset
    Button (290,326 91x30), "HALT"
        tap vAxis.bHalt
    Textfield (199,84 66x20), "%.2f", text variable: vAxis.rVel
        OnMouseDown: write the text variable via Default
    Label (157,86 36x22), "VEL"
    Textfield (62,99 66x20), "%.2f", text variable: vAxis.rPos
        OnMouseDown: write the text variable via Default
    Label (20,101 36x22), "POS"
    Textfield (199,154 66x20), "%.2f", text variable: vAxis.rJerk
        OnMouseDown: write the text variable via Default
    Label (157,156 36x22), "JERK"
    Textfield (199,118 66x20), "%.2f", text variable: vAxis.rAcc
        OnMouseDown: write the text variable via Default
    Label (157,120 36x22), "ACC"
    Button (13,54 55x30), "JOG +"
        tap vAxis.bJogPos
    Button (78,54 55x30), "JOG -"
        tap vAxis.bJogNeg
    Button (19,130 110x30), "GO ABS"
        OnMouseDown: execute { vAXIS.bMoveABS:=TRUE; }
    Textfield (61,184 66x20), "%.2f", text variable: vAxis.Dist
        OnMouseDown: write the text variable via Default
    Label (19,186 36x22), "DIST"
    Button (18,215 110x30), "GO REL"
        OnMouseDown: execute { vAXIS.bMoveRel:=TRUE; }
    Rectangle (16,15 99x30), "%s", text variable: vAxis.sName
    Button (169,39 98x15), "SET"
        tap vAxis.bSetPosition
    Button (17,269 110x30), "OPEN"
        OnMouseDown: execute { vAXIS.bOPEN:=TRUE;  vAXIS.bCLOSE:=FALSE; }
    Button (16,312 110x30), "CLOSE"
        OnMouseDown: execute { vAXIS.bCLOSE:=TRUE; vAXIS.bOPEN:=FALSE; }
    Lamp1 (138,263 40x45), variable: vAxis.bLIMIT_OPENED, style: Lamp-Lamp1-Yellow
    Lamp1 (137,308 40x45), variable: vAxis.bLIMIT_CLOSED, style: Lamp-Lamp1-Yellow
    Rectangle (15,350 110x28), "%s", text variable: vAxis.sAXIS_STATE
    Button (186,270 24x26)
        toggle vAxis.bLIMIT_OPENED
    Button (186,313 24x26)
        toggle vAxis.bLIMIT_CLOSED
    Button (290,364 91x30), "HOME"
        OnMouseDown: execute { vAxis.bHOME:=TRUE; }
    DipSwitch (224,365 30x30), variable: vAxis.bHOME_DIR, behaviour: TOGGLE, style: Switch-DipSwitch-Gray
    Lamp1 (260,368 25x34), variable: vAxis.bHOMED, style: Lamp-Lamp1-Blue
    Lamp1 (145,352 26x28), variable: vAxis.bSTATE_ERROR;, style: Lamp-Lamp1-Red
END_VISUALIZATION

// ---- POUs/EVENT_LOGGER/vEVENT_LOGGER.TcVIS
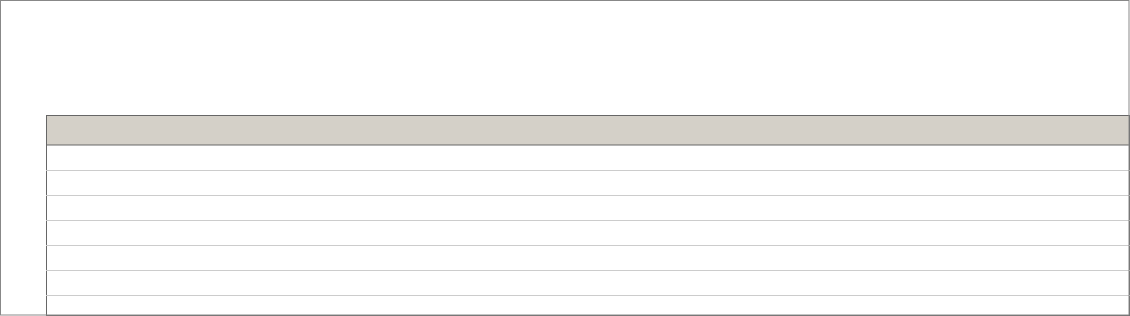
VISUALIZATION vEVENT_LOGGER  // 1130x316
    Table (46,115 1084x201), data array: fbEventLogger.EventBuffer
        p3854506369: fbEventLogger.EventBuffer[INDEX].eEventType
        p1892666644: fbEventLogger.EventBuffer[INDEX].eEventSeverity
        p338671338: fbEventLogger.EventBuffer[INDEX].nEventIdentity
        p2170511999: fbEventLogger.EventBuffer[INDEX].sEventName
        p3723444502: fbEventLogger.EventBuffer[INDEX].sEventText
        p1218418051: fbEventLogger.EventBuffer[INDEX].dtTimestamp
END_VISUALIZATION

// ---- POUs/PISTONS/vPISTONS.TcVIS
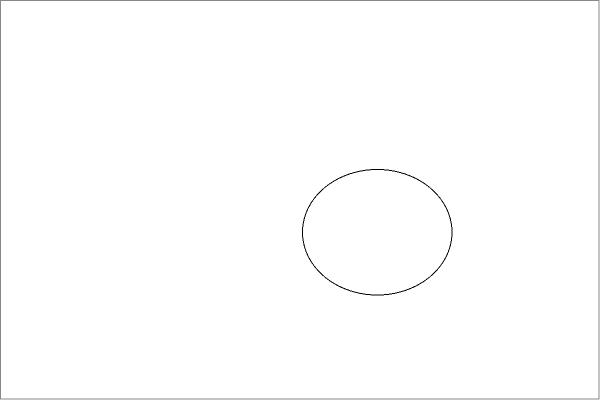
VISUALIZATION vPISTONS  // 600x400
    Ellipse (302,169 150x126)
END_VISUALIZATION

// ---- POUs/STATIONS/vSEPARATE.TcVIS
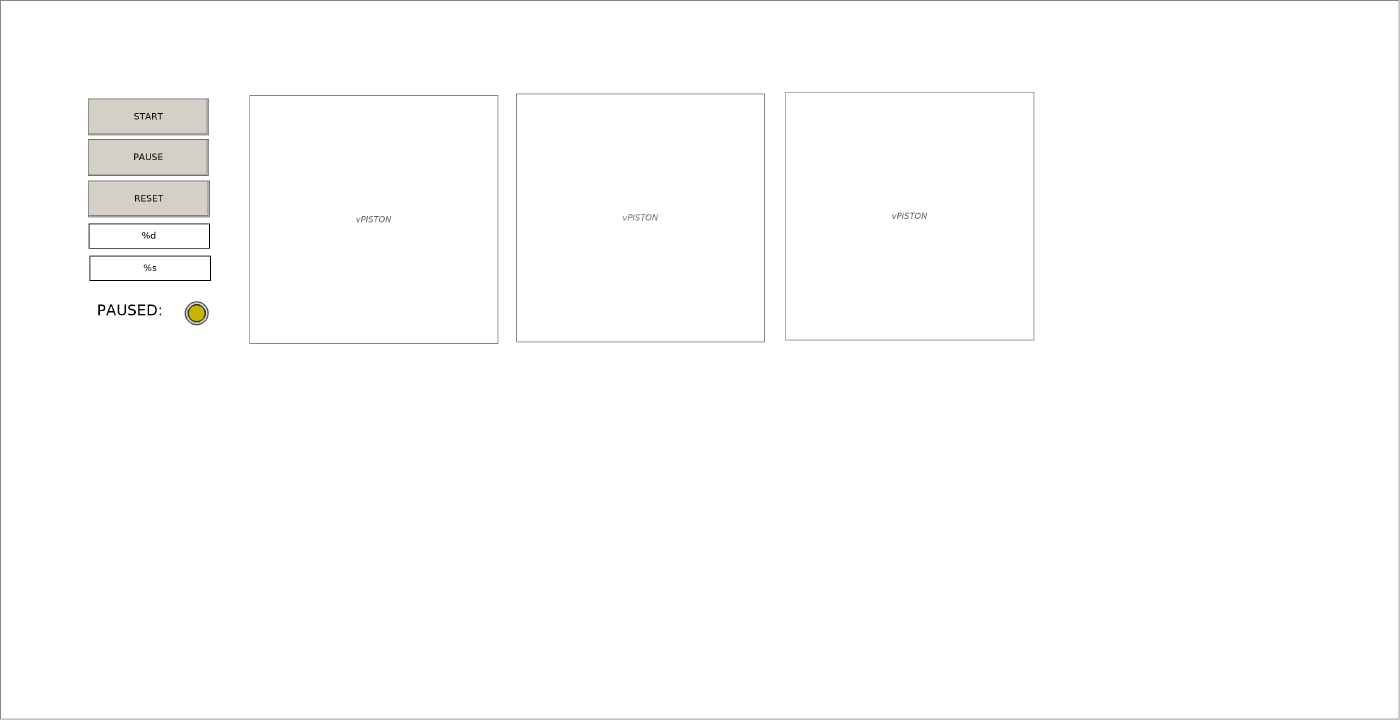
VISUALIZATION vSEPARATE  // 1690x870
VAR_IN_OUT
	vSEPARATE: FB_SEPARATE;
END_VAR
    Frame (301,115 300x300)
        shows vPISTON(PIST1 := vFEEDER.fbPIST1)
    Frame (623,113 300x300)
        shows vPISTON(PIST1 := vFEEDER.fbPIST2)
    Frame (948,111 300x300)
        shows vPISTON(PIST1 := vFEEDER.fbPIST3)
    Frame (87,109 200x360)
        shows vSTATION_CONTROLLER(vSTATION := vFEEDER)
END_VISUALIZATION

// ---- POUs/STATIONS/vSTATION_CONTROLLER.TcVIS
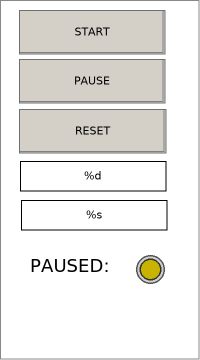
VISUALIZATION vSTATION_CONTROLLER  // 200x360
VAR_IN_OUT
	vSTATION : FB_STATION;
END_VAR
    Button (19,10 146x44), "START"
        OnMouseClick: execute { vSTATION.bSTART:=TRUE; }
    Button (19,109 147x44), "RESET"
        OnMouseClick: execute { vSTATION.bRESET:=TRUE; }
    Rectangle (20,161 146x30), "%d", text variable: vSTATION.iSTATION_STATE
    Rectangle (21,200 146x30), "%s", text variable: vSTATION.sSTATION_STATE
    Button (19,59 146x44), "PAUSE"
        toggle vSTATION.bPAUSE
    Lamp1 (134,248 33x43), variable: vSTATION.bPAUSE, style: Lamp-Lamp1-Yellow
    Label (26,251 88x30), "PAUSED:"
END_VISUALIZATION

// ---- VISUs/vCOMM.TcVIS
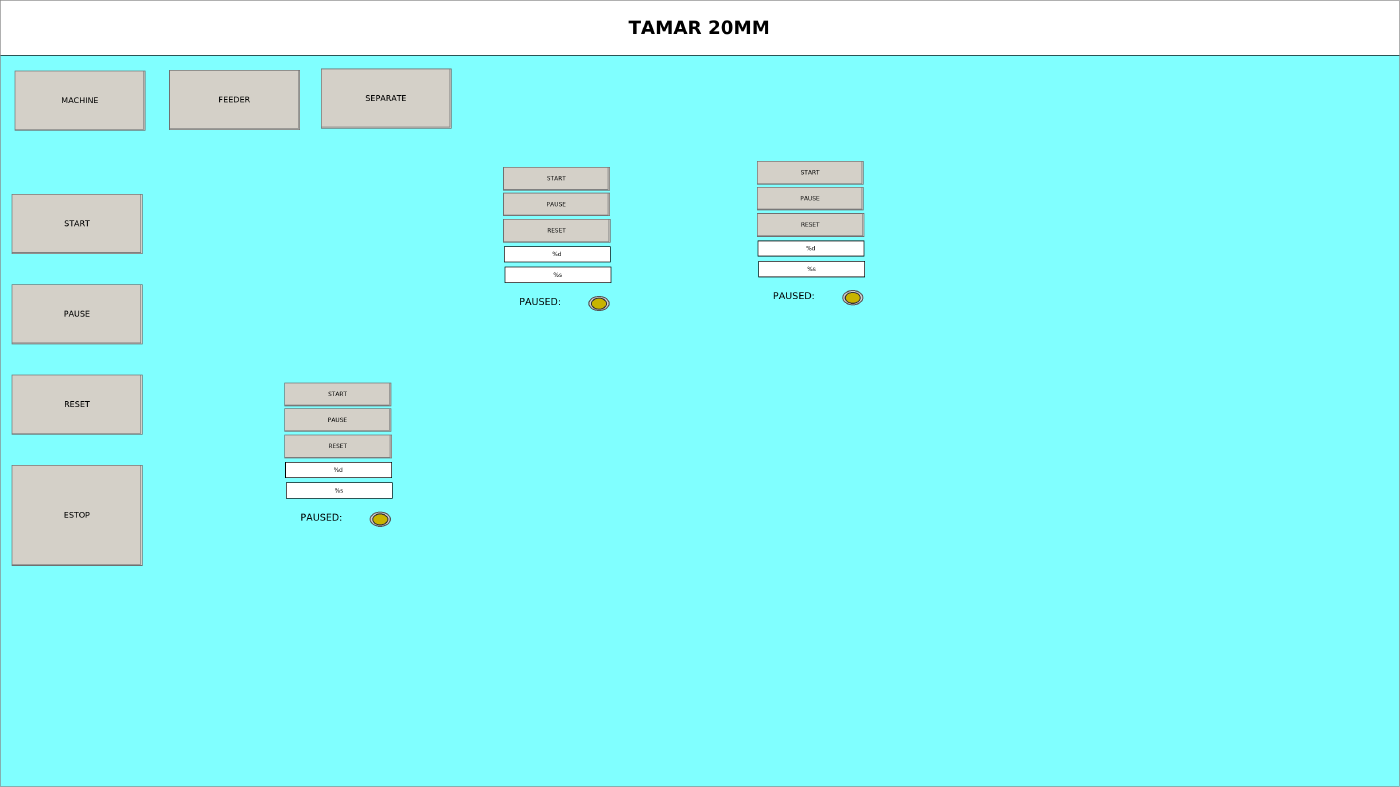
VISUALIZATION vCOMM  // 1920x1080
    Button (16,266 179x82), "START"
        OnMouseClick: FrameSelectionChange Selection=SelectedFrame=57b8a836-bac6-4cd4-9f68-9082885f5745, GlobSel=AssignType=Directly, SelType=Locally
    Rectangle (-3,-1 1924x77), "TAMAR 20MM"
    Button (16,390 179x82), "PAUSE"
        OnMouseClick: FrameSelectionChange Selection=SelectedFrame=57b8a836-bac6-4cd4-9f68-9082885f5745, GlobSel=AssignType=Directly, SelType=Locally
    Button (16,514 179x82), "RESET"
        OnMouseClick: FrameSelectionChange Selection=SelectedFrame=57b8a836-bac6-4cd4-9f68-9082885f5745, GlobSel=AssignType=Directly, SelType=Locally
    Button (16,638 179x138), "ESTOP"
        OnMouseClick: FrameSelectionChange Selection=SelectedFrame=57b8a836-bac6-4cd4-9f68-9082885f5745, GlobSel=AssignType=Directly, SelType=Locally
    Frame (278,203 1690x870)
        shows vMACHINE()
        shows vFEEDER(vFEEDER := fbFEEDER)
        shows vSEPARATE(vSEPARATE1 := fbSEPARATE1, vSEPARATE2 := fbSEPARATE2)
    Button (232,96 179x82), "FEEDER"
        OnMouseClick: FrameSelectionChange Selection=SelectedFrame=00e59953-e4a5-4fe1-b8af-e2191fac8d98, Selection=1, GlobSel=AssignType=Directly, SelType=Locally
    Button (20,97 179x82), "MACHINE"
        OnMouseClick: FrameSelectionChange Selection=SelectedFrame=00e59953-e4a5-4fe1-b8af-e2191fac8d98, GlobSel=AssignType=Directly, SelType=Locally
    Button (440,94 179x82), "SEPARATE"
        OnMouseClick: FrameSelectionChange Selection=SelectedFrame=00e59953-e4a5-4fe1-b8af-e2191fac8d98, Selection=2, GlobSel=AssignType=Directly, SelType=Locally
END_VISUALIZATION

// ---- VISUs/vMACHINE.TcVIS
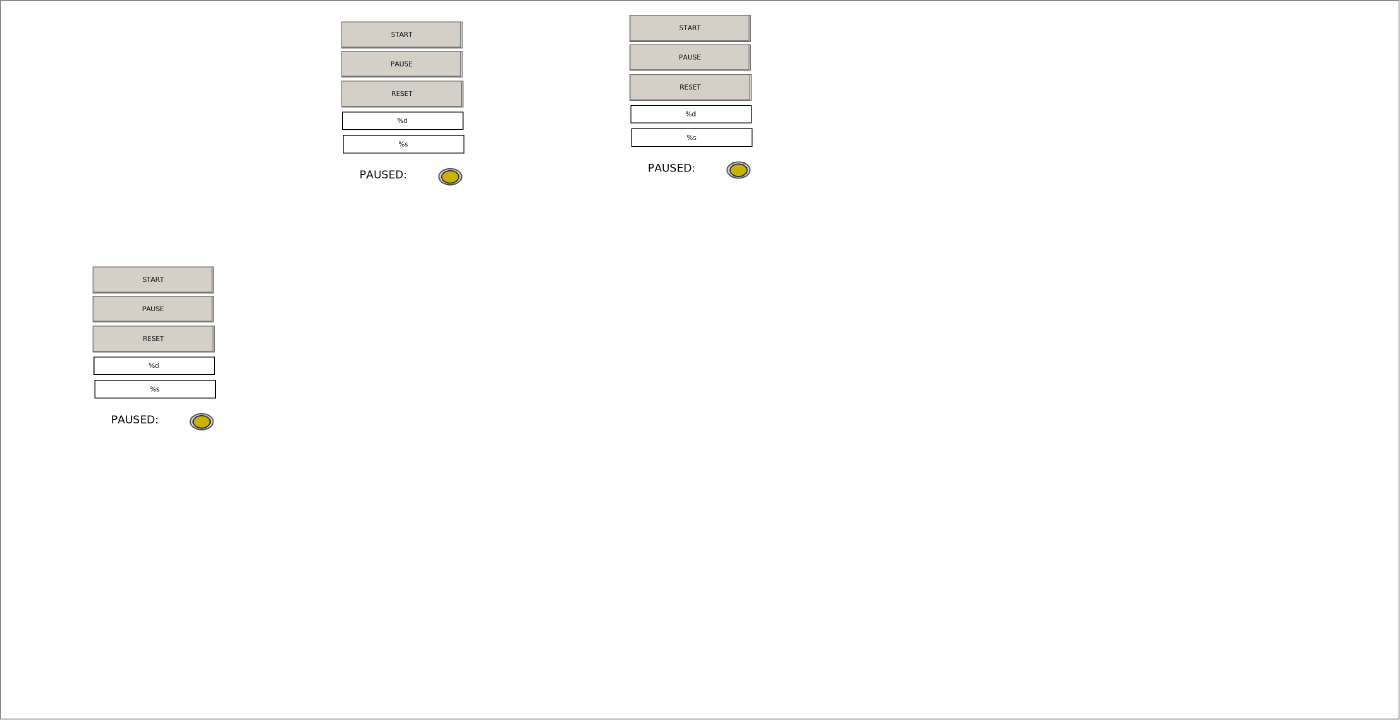
VISUALIZATION vMACHINE  // 1690x870
    Frame (93,315 200x260)
        shows vSTATION_CONTROLLER(vSTATION := fbFEEDER)
    Frame (393,19 200x260)
        shows vSTATION_CONTROLLER(vSTATION := fbSEPARATE1)
    Frame (741,11 200x260)
        shows vSTATION_CONTROLLER(vSTATION := fbSEPARATE2)
END_VISUALIZATION
